TYPE FsT_TypeClass : __SYSTEM.TYPE_CLASS; END_TYPE

(* stored: Version 1.1.0.1, ProductVersion 3.1.4024.4
   DUT FsT_TypeClass: Id {fd2b70ec-57ea-4e44-912e-67ab95a36604} *)
